//==================================================================================================
//							Beckhoff Automation Poland
//									18.04.2018
//	Struktura zawierajaca I/O odpowiedniego bloku
//  v1.0	|| TC v 3.1.4022.16		|| - pierwsza wersja
//==================================================================================================
TYPE ST_MCHomeIO:
STRUCT
	bExecute						: BOOL;								// Rising edge executes cmd
	lrPosition						: LREAL					:= DEFAULT_HOME_POSITION;
	eHomingMode						: Tc2_MC2.MC_HomingMode;
	eBufferMode						: Tc2_MC2.MC_BufferMode;
	stOptions						: Tc2_MC2.ST_HomingOptions;
	bCalibrationCam					: BOOL;
	bDone							: BOOL;
	bBusy							: BOOL;
	bActive							: BOOL;
	bCommandAborted					: BOOL;
	bError							: BOOL;
	udiErrorID						: UDINT;
END_STRUCT
END_TYPE

(* stored: Version 1.1.0.1, ProductVersion 3.1.4026.13, FileIdentifier fdb096913c68fefb14feb6d39e721d31c27ac8cf, FileSignature 8e003493f3001f42f60c883b34a5e3c3403261fb51f18233eaa1c76da7887df11b42ca481f4e3d8dc746cc975fab9d445b4985954ce9ba0abc44f5d9440b94a48bc8555e5f241f6f1c8247e11673848a2d2f931406f855d4ff7f66471998ed5660c89c0c43b49b3878f1daff8dbabda75873a7a5ebbea4dc993653d7a9301f3fd58896983089569028413fe113d21c6ec843c98abf1cda205d462b91800ef49b65c7e28e7c14cec07617bcf1728acfa88b700195889038715161980e1912c3cff8da9d6a529da5c426f52cbbb48e19687e0f6c29e4f7b45ae930bf38d720fbd5a894ff3e84de1ca9dafa928c5d48e0c44900d16b0bdb60767856efbd0d54a12f
   DUT ST_MCHomeIO: Id {f0ac6427-a2cd-40f7-b604-aaf9bca4868c} *)
